FUNCTION_BLOCK PalletID_Name
VAR_INPUT
	CounterBox	: USINT;
	
	sYear		: STRING;
	sMonth		: STRING;
	sDate		: STRING;
	sHour		: STRING;
	sMinutes	: STRING;
	sSeconds	: STRING;
	PalletNumber: STRING(2);
	LineNumber	: STRING(2);
END_VAR
VAR_OUTPUT PERSISTENT
	PalletID	: STRING;
END_VAR
VAR
	Timer: TON;
END_VAR

VAR PERSISTENT
	PalletData: STRING;
	SeqIndex: INT;
END_VAR

PalletID:=PalletData; // Assign nilai dari variabel PalletData ke variabel PalletID

CASE SeqIndex OF // Memulai blok pemilihan kasus berdasarkan nilai SeqIndex
	0: // Kasus saat SeqIndex = 0
		IF (CounterBox=1) THEN // Jika nilai CounterBox adalah 1
			SeqIndex:=10; // Ganti nilai SeqIndex menjadi 10
		END_IF // Selesai kondisi IF
	10: // Kasus saat SeqIndex = 10
		PalletData:=CONCAT(PalletNumber,CONCAT(sHour,CONCAT(sMinutes,CONCAT(sSeconds,CONCAT(sDate,CONCAT(sMonth,sYear)))))); // Gabungkan nilai-nilai string yang diberikan dalam variabel PalletData
		SeqIndex:=20; // Ganti nilai SeqIndex menjadi 20
	20: // Kasus saat SeqIndex = 20
		IF NOT (CounterBox=1) THEN // Jika nilai CounterBox bukan 1
			SeqIndex:=0; // Ganti nilai SeqIndex menjadi 0
		END_IF // Selesai kondisi IF
END_CASE // Selesai blok pemilihan kasus

END_FUNCTION_BLOCK

(* stored: Version 1.1.0.1, ProductVersion 3.1.4024.6
   POU PalletID_Name: Id {10a30c02-f6db-4cc0-8861-05e0a84d5e94}, SpecialFunc None *)
